INTERFACE I_AxDriveBase EXTENDS __SYSTEM.IQueryInterface

PROPERTY PUBLIC rAxDrive : REFERENCE TO AxDriveBase
GET
END_GET
END_PROPERTY

END_INTERFACE

(* stored: Version 1.1.0.1, ProductVersion 3.1.4024.4
   Itf I_AxDriveBase: Id {bd294a7b-9420-4419-8749-42aea727b934}
   Property rAxDrive: Id {1c3d979c-3af3-43ea-9f00-ede3a090d6fe}
   Get Get: Id {5ef96e38-26fe-4ae6-8dd2-f6f60766037c} *)
